// TwinCAT 3 PLC project TrafficLights_PLC
// ProgramVersion: 3.1.4024.0
// libraries:
//   Tc2_Standard, * (Beckhoff Automation GmbH)
//   Tc2_System, * (Beckhoff Automation GmbH)
//   Tc3_Module, * (Beckhoff Automation GmbH)
//   VisuSymbols,3.5.10.0,System
// project tree:
//   DUTs/ E_TrafficState.TcDUT
//   / GlobalTextList.TcGTLO, PlcTask.TcTTO, Visualization Manager.TcVMO (not stored)
//   POUs/ MAIN.TcPOU
//   VISUs/ Visualization.TcVIS

CONFIGURATION TrafficLights_PLC
    RESOURCE PLC ON TwinCAT3
        TASK PlcTask(INTERVAL := T#10ms, PRIORITY := 20);
        PROGRAM MAIN WITH PlcTask : MAIN;
    END_RESOURCE
END_CONFIGURATION

// ---- DUTs/E_TrafficState.TcDUT
{attribute 'qualified_only'}
TYPE E_TrafficState :
(
    STATE_RED       := 0,
    STATE_RED_AMBER := 1,
    STATE_GREEN     := 2,
    STATE_AMBER     := 3
);
END_TYPE

// ---- POUs/MAIN.TcPOU
PROGRAM MAIN
VAR
    (* State machine *)
    eState          : E_TrafficState := E_TrafficState.STATE_RED;

    (* TwinCAT timer *)
    tonTimer        : TON;
    tDuration       : TIME := T#5S;   (* current phase duration *)

    (* Light outputs — wire these to real I/O or watch in simulation *)
    bRed            : BOOL;
    bAmber          : BOOL;
    bGreen          : BOOL;
END_VAR

(* ── Run the timer ────────────────────────────────────────── *)
tonTimer(IN := NOT tonTimer.Q, PT := tDuration);

(* ── State machine ───────────────────────────────────────── *)
IF tonTimer.Q THEN

    CASE eState OF

        E_TrafficState.STATE_RED:
            eState    := E_TrafficState.STATE_RED_AMBER;
            tDuration := T#2S;

        E_TrafficState.STATE_RED_AMBER:
            eState    := E_TrafficState.STATE_GREEN;
            tDuration := T#5S;

        E_TrafficState.STATE_GREEN:
            eState    := E_TrafficState.STATE_AMBER;
            tDuration := T#2S;

        E_TrafficState.STATE_AMBER:
            eState    := E_TrafficState.STATE_RED;
            tDuration := T#5S;

    END_CASE

END_IF

(* ── Set outputs based on current state ─────────────────── *)
bRed   := (eState = E_TrafficState.STATE_RED)
       OR (eState = E_TrafficState.STATE_RED_AMBER);

bAmber := (eState = E_TrafficState.STATE_RED_AMBER)
       OR (eState = E_TrafficState.STATE_AMBER);

bGreen := (eState = E_TrafficState.STATE_GREEN);

END_PROGRAM

// ---- VISUs/Visualization.TcVIS
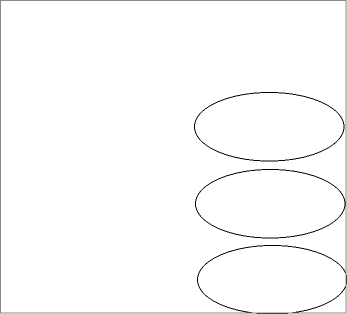
VISUALIZATION Visualization  // 347x314
    Ellipse (194,92 150x69), colour toggle: MAIN.bRed
    Ellipse (195,169 150x69), colour toggle: MAIN.bAmber
    Ellipse (197,245 150x69), colour toggle: MAIN.bGreen
END_VISUALIZATION
